{attribute 'qualified_only'}
{attribute 'strict'}
TYPE E_ReportType :
(
	None := 0,
    PumpCalibration := 1,
    SystemSettings := 2,
    PostRun := 3,
    LinearMotors := 4,
    Recipe := 5
);
END_TYPE

(* stored: Version 1.1.0.1, ProductVersion 3.1.4024.15
   DUT E_ReportType: Id {ded1da90-1ca9-4afa-97aa-91829e31cba3} *)
